(* IEC 61131-3 sources: ladder-web-ide/spikes/modelo/preset25, 22 files *)

(* ---- variante_a_pv13_base.st ---- *)
(* Variante A -- BASELINE do preset25 (spikes/modelo/NOTAS.md, "Experimento
   BLINK"). E o mesmo desenho/ST de spikes/modelo/blink_ladder.st (PV=13),
   reproduzido aqui como ponto de partida da matriz, para todas as variantes
   ficarem juntas e serem medidas pelo mesmo medir.py. Ver RESULTADO.md para
   a tabela comparativa.

   Ladder (ASCII; "%" = ramo paralelo na linha 1):

   Rung 1 (pulso, oscilador de 1 ciclo):
   ====|/pulso|==================( pulso )====

   Rung 2 (contador):
   ====|pulso|===+==[ CTU PV=13 ]===saida=atingiu====
                 %
                 +--|reset_ctu|--+   (ramo linha 1, alimenta R)

   Rung 3 (agenda reset, MINIMO de 1 ciclo de atraso -- e o proprio Q lido
           1 ciclo depois, por construcao: nao ha como um CTU usar seu
           proprio Q como R na MESMA chamada -- ver RESULTADO.md, prova):
   ====|atingiu|=================( reset_ctu )====

   Rung 4 (instantaneo de led, evita auto-cancelamento SET/RESET no mesmo
           scan -- ver NOTAS.md, "Risco descoberto no experimento"):
   ====|led|======================( led_estava_aceso )====

   Rung 5 (liga led):
   ====|atingiu|==|/led_estava_aceso|========(S led )====

   Rung 6 (desliga led):
   ====|atingiu|==|led_estava_aceso|=========(R led )====

   Rung 7 (botao, igual ao blink.st original):
   ====|botao|====================(S led )====

   ST derivado (ordem de leitura = ordem de execucao):
     pulso := NOT pulso;
     ctu0(CU := pulso, R := reset_ctu, PV := 13);
     atingiu := ctu0.Q;
     reset_ctu := atingiu;
     led_estava_aceso := led;
     IF atingiu AND NOT led_estava_aceso THEN led := TRUE; END_IF;
     IF atingiu AND led_estava_aceso THEN led := FALSE; END_IF;
     IF botao THEN led := TRUE; END_IF;

   Sem acentos: ASCII puro para o compilador. *)

PROGRAM prog0
  VAR
    botao AT %IX0.0 : BOOL;
    led   AT %QX0.0 : BOOL;
  END_VAR
  VAR
    pulso            : BOOL;
    reset_ctu        : BOOL;
    atingiu          : BOOL;
    led_estava_aceso : BOOL;
    ctu0             : CTU;
  END_VAR

  (* Rung 1 *)
  pulso := NOT pulso;

  (* Rung 2 *)
  ctu0(CU := pulso, R := reset_ctu, PV := 13);
  atingiu := ctu0.Q;

  (* Rung 3 -- reset com o atraso MINIMO possivel (1 scan) *)
  reset_ctu := atingiu;

  (* Rung 4 -- instantaneo de led *)
  led_estava_aceso := led;

  (* Rung 5 *)
  IF atingiu AND NOT led_estava_aceso THEN
    led := TRUE;
  END_IF;

  (* Rung 6 *)
  IF atingiu AND led_estava_aceso THEN
    led := FALSE;
  END_IF;

  (* Rung 7 *)
  IF botao THEN
    led := TRUE;
  END_IF;
END_PROGRAM

CONFIGURATION Config0
  RESOURCE Res0 ON PLC
    TASK task0(INTERVAL := T#20ms, PRIORITY := 0);
    PROGRAM instance0 WITH task0 : prog0;
  END_RESOURCE
END_CONFIGURATION

(* ---- variante_b_pv12.st ---- *)
(* Variante B -- mesmo desenho da variante A, PV=12 em vez de 13 (mesma
   tentativa "PV diferente" ja medida em spikes/modelo/blink_ladder_pv12.st,
   reproduzida aqui para entrar na mesma bateria de medicao de 200 ciclos /
   3 padroes de %IX0.0 do preset25). Ver RESULTADO.md.

   Ladder identico ao da variante A (variante_a_pv13_base.st), so troca
   PV:=13 por PV:=12 no rung 2. ST derivado idem, com PV:=12. *)

PROGRAM prog0
  VAR
    botao AT %IX0.0 : BOOL;
    led   AT %QX0.0 : BOOL;
  END_VAR
  VAR
    pulso            : BOOL;
    reset_ctu        : BOOL;
    atingiu          : BOOL;
    led_estava_aceso : BOOL;
    ctu0             : CTU;
  END_VAR

  (* Rung 1 *)
  pulso := NOT pulso;

  (* Rung 2 -- unica diferenca frente a variante A: PV=12 *)
  ctu0(CU := pulso, R := reset_ctu, PV := 12);
  atingiu := ctu0.Q;

  (* Rung 3 *)
  reset_ctu := atingiu;

  (* Rung 4 *)
  led_estava_aceso := led;

  (* Rung 5 *)
  IF atingiu AND NOT led_estava_aceso THEN
    led := TRUE;
  END_IF;

  (* Rung 6 *)
  IF atingiu AND led_estava_aceso THEN
    led := FALSE;
  END_IF;

  (* Rung 7 *)
  IF botao THEN
    led := TRUE;
  END_IF;
END_PROGRAM

CONFIGURATION Config0
  RESOURCE Res0 ON PLC
    TASK task0(INTERVAL := T#20ms, PRIORITY := 0);
    PROGRAM instance0 WITH task0 : prog0;
  END_RESOURCE
END_CONFIGURATION

(* ---- variante_c_pv25.st ---- *)
(* Variante C -- mesmo desenho da variante A, PV=25 (o valor "obvio" -- PV
   igual ao limite de contador.st -- citado no enunciado como tentativa a
   medir). Previsao analitica (RESULTADO.md, prova do periodo minimo
   T=2*PV): com CU alternando 1 vez por ciclo (borda a cada 2 ciclos) e reset
   consumindo 1 ciclo, o periodo minimo entre disparos de `atingiu` e
   2*25=50 ciclos -- 2x mais lento que os 25 ciclos de blink.st, nao um
   candidato melhor que PV=13. Medido aqui para confirmar. *)

PROGRAM prog0
  VAR
    botao AT %IX0.0 : BOOL;
    led   AT %QX0.0 : BOOL;
  END_VAR
  VAR
    pulso            : BOOL;
    reset_ctu        : BOOL;
    atingiu          : BOOL;
    led_estava_aceso : BOOL;
    ctu0             : CTU;
  END_VAR

  (* Rung 1 *)
  pulso := NOT pulso;

  (* Rung 2 -- unica diferenca frente a variante A: PV=25 *)
  ctu0(CU := pulso, R := reset_ctu, PV := 25);
  atingiu := ctu0.Q;

  (* Rung 3 *)
  reset_ctu := atingiu;

  (* Rung 4 *)
  led_estava_aceso := led;

  (* Rung 5 *)
  IF atingiu AND NOT led_estava_aceso THEN
    led := TRUE;
  END_IF;

  (* Rung 6 *)
  IF atingiu AND led_estava_aceso THEN
    led := FALSE;
  END_IF;

  (* Rung 7 *)
  IF botao THEN
    led := TRUE;
  END_IF;
END_PROGRAM

CONFIGURATION Config0
  RESOURCE Res0 ON PLC
    TASK task0(INTERVAL := T#20ms, PRIORITY := 0);
    PROGRAM instance0 WITH task0 : prog0;
  END_RESOURCE
END_CONFIGURATION

(* ---- variante_d_pv13_reset_atrasado.st ---- *)
(* Variante D -- PV=13, reset com 1 ciclo de atraso EXTRA (2 scans no total,
   em vez do minimo de 1 -- ver variante A) frente ao momento em que
   `atingiu` fica verdadeiro. Testa a celula da matriz "reset imediato
   (minimo possivel, variante A) vs atrasado" pedida no enunciado.

   Para conseguir um segundo scan de atraso sem tocar no elemento `ctu` (que
   so aceita R vindo de um caminho de contatos), uso DOIS estagios de
   bobina -- mas a ORDEM dos rungs importa (isto foi corrigido depois de
   medir: a primeira versao desta variante, com os dois rungs na ordem
   "contrario", nao acrescentava atraso nenhum -- ver NOTA DE MEDICAO no
   fim deste comentario):

     Rung 3 (ANTES do estagio 1): reset_ctu := reset_estagio1
       -- le reset_estagio1 como estava NO INICIO deste scan (o rung
       seguinte ainda nao o atualizou), ou seja o valor que o rung 4
       escreveu no scan ANTERIOR.
     Rung 4 (DEPOIS): reset_estagio1 := atingiu
       -- atualiza com o `atingiu` fresco deste mesmo scan.

   Com essa ordem: reset_estagio1(n) = atingiu(n); reset_ctu(n) =
   reset_estagio1(n-1) [valor pre-atualizacao] = atingiu(n-1). O `R` usado
   pela chamada do CTU no scan n+1 e reset_ctu(n) = atingiu(n-1) -- 2 scans
   de atraso frente a atingiu(n), 1 scan a mais que a variante A (que da
   R(n+1) = atingiu(n)).

   Ladder (ASCII):

   Rung 1 (pulso):
   ====|/pulso|==================( pulso )====

   Rung 2 (contador, mesmo desenho da variante A):
   ====|pulso|===+==[ CTU PV=13 ]===saida=atingiu====
                 %
                 +--|reset_ctu|--+

   Rung 3 (le o estagio 1 ANTES dele ser atualizado neste mesmo scan --
           e o que da o segundo scan de atraso):
   ====|reset_estagio1|===========( reset_ctu )====

   Rung 4 (so agora atualiza o estagio 1 com o `atingiu` fresco):
   ====|atingiu|=================( reset_estagio1 )====

   Rung 5 (instantaneo de led, igual a variante A):
   ====|led|======================( led_estava_aceso )====

   Rung 6 (liga led):
   ====|atingiu|==|/led_estava_aceso|========(S led )====

   Rung 7 (desliga led):
   ====|atingiu|==|led_estava_aceso|=========(R led )====

   Rung 8 (botao):
   ====|botao|====================(S led )====

   ST derivado:
     pulso := NOT pulso;
     ctu0(CU := pulso, R := reset_ctu, PV := 13);
     atingiu := ctu0.Q;
     reset_ctu := reset_estagio1;
     reset_estagio1 := atingiu;
     led_estava_aceso := led;
     IF atingiu AND NOT led_estava_aceso THEN led := TRUE; END_IF;
     IF atingiu AND led_estava_aceso THEN led := FALSE; END_IF;
     IF botao THEN led := TRUE; END_IF;

   NOTA DE MEDICAO (achado no proprio processo de montar esta variante, nao
   so no experimento original): a primeira tentativa de escrever este atraso
   extra colocou "reset_estagio1 := atingiu" ANTES de "reset_ctu :=
   reset_estagio1", isto e, deixou o valor fresco de `atingiu` atravessar os
   dois estagios NO MESMO SCAN (rung3 grava reset_estagio1(n)=atingiu(n);
   rung4, logo em seguida, ja le esse valor fresco e grava
   reset_ctu(n)=atingiu(n) -- zero atraso ADICIONAL, resultado identico ao
   da variante A). So a ordem escrita acima (ler o estagio seguinte ANTES de
   atualizar o anterior) de fato empurra 1 scan a mais -- e a mesma logica,
   inversa, de por que a variante A ja e o atraso MINIMO possivel (rung do
   reset depois do rung do CTU): o numero de scans de atraso de uma cadeia
   de bobinas depende de QUAL lado da cadeia e lido antes do outro ser
   escrito, nao so de quantos estagios existem. Medido com medir.py: a
   PRIMEIRA versao (sem atraso extra de fato) deu os MESMOS 22/22/21
   divergencias da variante A; esta versao corrigida e a que aparece na
   tabela de RESULTADO.md como "variante D". *)

PROGRAM prog0
  VAR
    botao AT %IX0.0 : BOOL;
    led   AT %QX0.0 : BOOL;
  END_VAR
  VAR
    pulso            : BOOL;
    reset_estagio1   : BOOL;
    reset_ctu        : BOOL;
    atingiu          : BOOL;
    led_estava_aceso : BOOL;
    ctu0             : CTU;
  END_VAR

  (* Rung 1 *)
  pulso := NOT pulso;

  (* Rung 2 *)
  ctu0(CU := pulso, R := reset_ctu, PV := 13);
  atingiu := ctu0.Q;

  (* Rung 3 -- le reset_estagio1 ANTES do rung 4 atualiza-lo (2o scan de atraso) *)
  reset_ctu := reset_estagio1;

  (* Rung 4 -- so agora atualiza com o atingiu fresco deste scan *)
  reset_estagio1 := atingiu;

  (* Rung 5 *)
  led_estava_aceso := led;

  (* Rung 6 *)
  IF atingiu AND NOT led_estava_aceso THEN
    led := TRUE;
  END_IF;

  (* Rung 7 *)
  IF atingiu AND led_estava_aceso THEN
    led := FALSE;
  END_IF;

  (* Rung 8 *)
  IF botao THEN
    led := TRUE;
  END_IF;
END_PROGRAM

CONFIGURATION Config0
  RESOURCE Res0 ON PLC
    TASK task0(INTERVAL := T#20ms, PRIORITY := 0);
    PROGRAM instance0 WITH task0 : prog0;
  END_RESOURCE
END_CONFIGURATION

(* ---- variante_e_pv13_toggle_paralelo.st ---- *)
(* Variante E -- PV=13, mesmo contador da variante A, mas o `led` alterna
   por um UNICO rung combinacional (ramo paralelo), nao por par SET/RESET.
   Testa a celula da matriz "toggle por ramo paralelo com bobina simples:
   led := (atingiu AND NOT led) OR (NOT atingiu AND led)".

   Motivo de interesse independente da fase: este desenho substitui os
   rungs 4/5/6 da variante A (instantaneo + par SET/RESET) por 1 rung so,
   eliminando de saida o risco de auto-cancelamento no mesmo scan descrito
   em NOTAS.md (nao ha dois rungs escrevendo o mesmo bit no mesmo scan) --
   `led_estava_aceso` deixa de ser necessario. Verifica-se aqui se isso muda
   a contagem/posicao das divergencias de fase (nao deveria: e uma troca de
   MECANISMO de toggle, nao do periodo do CTU).

   Ladder (ASCII):

   Rung 1 (pulso):
   ====|/pulso|==================( pulso )====

   Rung 2 (contador, igual a variante A):
   ====|pulso|===+==[ CTU PV=13 ]===saida=atingiu====
                 %
                 +--|reset_ctu|--+

   Rung 3 (agenda reset, igual a variante A):
   ====|atingiu|=================( reset_ctu )====

   Rung 4 (toggle combinacional -- DOIS caminhos em paralelo que se juntam
           na mesma bobina `led`; nenhum SET/RESET):
   ====|atingiu|==|/led|====+==================( led )====
   ====|/atingiu|==|led|====+

   Rung 5 (botao, igual a variante A):
   ====|botao|====================(S led )====

   ST derivado (a bobina comum de um rung com ramo paralelo e o OU dos
   caminhos serie -- aqui exatamente a expressao do enunciado):
     pulso := NOT pulso;
     ctu0(CU := pulso, R := reset_ctu, PV := 13);
     atingiu := ctu0.Q;
     reset_ctu := atingiu;
     led := (atingiu AND NOT led) OR (NOT atingiu AND led);
     IF botao THEN led := TRUE; END_IF; *)

PROGRAM prog0
  VAR
    botao AT %IX0.0 : BOOL;
    led   AT %QX0.0 : BOOL;
  END_VAR
  VAR
    pulso     : BOOL;
    reset_ctu : BOOL;
    atingiu   : BOOL;
    ctu0      : CTU;
  END_VAR

  (* Rung 1 *)
  pulso := NOT pulso;

  (* Rung 2 *)
  ctu0(CU := pulso, R := reset_ctu, PV := 13);
  atingiu := ctu0.Q;

  (* Rung 3 *)
  reset_ctu := atingiu;

  (* Rung 4 -- toggle por ramo paralelo, sem SET/RESET *)
  led := (atingiu AND NOT led) OR (NOT atingiu AND led);

  (* Rung 5 *)
  IF botao THEN
    led := TRUE;
  END_IF;
END_PROGRAM

CONFIGURATION Config0
  RESOURCE Res0 ON PLC
    TASK task0(INTERVAL := T#20ms, PRIORITY := 0);
    PROGRAM instance0 WITH task0 : prog0;
  END_RESOURCE
END_CONFIGURATION

(* ---- variante_f_pv13_pulso_inicial_true.st ---- *)
(* Variante F -- PV=13, mesmo desenho da variante A, so muda o valor
   INICIAL de `pulso` para TRUE em vez do default FALSE. Testa a celula da
   matriz "pulso inicial FALSE/TRUE".

   ACHADO A REGISTRAR (ver RESULTADO.md): o modelo grafico obrigatorio
   (spikes/modelo/modelo.ts, interface `Variavel`) NAO tem campo de valor
   inicial -- so `nome`, `tipo`, `endereco?`. Esta variante e expressavel em
   ST puro (`pulso : BOOL := TRUE;`, sintaxe valida de IEC 61131-3), mas NAO
   e desenhavel com o modelo de dados da grade tal como ele existe hoje: um
   editor Ladder que use esse modelo nao tem como o autor do diagrama pedir
   "essa variavel comeca em TRUE". Se esta variante fosse a vencedora,
   `Variavel` precisaria ganhar um campo tipo `valorInicial?: boolean` (so
   faz sentido para BOOL nao localizado; UINT e localizado ficam fora). Ela
   NAO e a vencedora (ver RESULTADO.md), entao o gap fica soh registrado,
   sem exigir mudanca no modelo.

   Ladder: identico a variante A (nao ha elemento grafico que represente
   "valor inicial"; a diferenca so aparece no ST). *)

PROGRAM prog0
  VAR
    botao AT %IX0.0 : BOOL;
    led   AT %QX0.0 : BOOL;
  END_VAR
  VAR
    pulso            : BOOL := TRUE; (* unica diferenca frente a variante A *)
    reset_ctu        : BOOL;
    atingiu          : BOOL;
    led_estava_aceso : BOOL;
    ctu0             : CTU;
  END_VAR

  (* Rung 1 *)
  pulso := NOT pulso;

  (* Rung 2 *)
  ctu0(CU := pulso, R := reset_ctu, PV := 13);
  atingiu := ctu0.Q;

  (* Rung 3 *)
  reset_ctu := atingiu;

  (* Rung 4 *)
  led_estava_aceso := led;

  (* Rung 5 *)
  IF atingiu AND NOT led_estava_aceso THEN
    led := TRUE;
  END_IF;

  (* Rung 6 *)
  IF atingiu AND led_estava_aceso THEN
    led := FALSE;
  END_IF;

  (* Rung 7 *)
  IF botao THEN
    led := TRUE;
  END_IF;
END_PROGRAM

CONFIGURATION Config0
  RESOURCE Res0 ON PLC
    TASK task0(INTERVAL := T#20ms, PRIORITY := 0);
    PROGRAM instance0 WITH task0 : prog0;
  END_RESOURCE
END_CONFIGURATION

(* ---- variante_g_pv13_ordem_invertida.st ---- *)
(* Variante G -- PV=13, mesmo desenho da variante A, mas o rung do CTU vem
   ANTES do rung que alterna `pulso` (ordem de leitura trocada). Testa a
   celula da matriz "rung de pulso antes/depois do rung do CTU".

   Com essa troca, o `CU` que o CTU le no scan N e o `pulso` como ficou no
   FIM do scan N-1 (o toggle deste scan so acontece DEPOIS, no rung
   seguinte) -- desloca a fase de leitura de `pulso` em 1 scan frente a
   variante A, analogo ao que um valor inicial diferente faria, mas via
   ordem de rung em vez de valor inicial (essa SIM e desenhavel no modelo
   grafico hoje: e so por o rung do contador antes do rung do oscilador na
   lista `rungs` do `Diagrama` -- nao exige nenhum campo novo).

   Ladder (ASCII; ordem trocada frente a variante A):

   Rung 1 (contador, agora primeiro):
   ====|pulso|===+==[ CTU PV=13 ]===saida=atingiu====
                 %
                 +--|reset_ctu|--+

   Rung 2 (pulso, agora depois):
   ====|/pulso|==================( pulso )====

   Rung 3 (agenda reset):
   ====|atingiu|=================( reset_ctu )====

   Rung 4 (instantaneo de led):
   ====|led|======================( led_estava_aceso )====

   Rung 5 (liga led):
   ====|atingiu|==|/led_estava_aceso|========(S led )====

   Rung 6 (desliga led):
   ====|atingiu|==|led_estava_aceso|=========(R led )====

   Rung 7 (botao):
   ====|botao|====================(S led )====

   ST derivado (so a ordem das duas primeiras atribuicoes muda frente a
   variante A):
     ctu0(CU := pulso, R := reset_ctu, PV := 13);
     atingiu := ctu0.Q;
     pulso := NOT pulso;
     reset_ctu := atingiu;
     led_estava_aceso := led;
     IF atingiu AND NOT led_estava_aceso THEN led := TRUE; END_IF;
     IF atingiu AND led_estava_aceso THEN led := FALSE; END_IF;
     IF botao THEN led := TRUE; END_IF; *)

PROGRAM prog0
  VAR
    botao AT %IX0.0 : BOOL;
    led   AT %QX0.0 : BOOL;
  END_VAR
  VAR
    pulso            : BOOL;
    reset_ctu        : BOOL;
    atingiu          : BOOL;
    led_estava_aceso : BOOL;
    ctu0             : CTU;
  END_VAR

  (* Rung 1 -- contador, ANTES do toggle de pulso (ordem trocada) *)
  ctu0(CU := pulso, R := reset_ctu, PV := 13);
  atingiu := ctu0.Q;

  (* Rung 2 -- pulso, agora depois *)
  pulso := NOT pulso;

  (* Rung 3 *)
  reset_ctu := atingiu;

  (* Rung 4 *)
  led_estava_aceso := led;

  (* Rung 5 *)
  IF atingiu AND NOT led_estava_aceso THEN
    led := TRUE;
  END_IF;

  (* Rung 6 *)
  IF atingiu AND led_estava_aceso THEN
    led := FALSE;
  END_IF;

  (* Rung 7 *)
  IF botao THEN
    led := TRUE;
  END_IF;
END_PROGRAM

CONFIGURATION Config0
  RESOURCE Res0 ON PLC
    TASK task0(INTERVAL := T#20ms, PRIORITY := 0);
    PROGRAM instance0 WITH task0 : prog0;
  END_RESOURCE
END_CONFIGURATION

(* ---- variante_h_pv12_reset_atrasado.st ---- *)
(* Variante D -- PV=13, reset com 1 ciclo de atraso EXTRA (2 scans no total,
   em vez do minimo de 1 -- ver variante A) frente ao momento em que
   `atingiu` fica verdadeiro. Testa a celula da matriz "reset imediato
   (minimo possivel, variante A) vs atrasado" pedida no enunciado.

   Para conseguir um segundo scan de atraso sem tocar no elemento `ctu` (que
   so aceita R vindo de um caminho de contatos), uso DOIS estagios de
   bobina -- mas a ORDEM dos rungs importa (isto foi corrigido depois de
   medir: a primeira versao desta variante, com os dois rungs na ordem
   "contrario", nao acrescentava atraso nenhum -- ver NOTA DE MEDICAO no
   fim deste comentario):

     Rung 3 (ANTES do estagio 1): reset_ctu := reset_estagio1
       -- le reset_estagio1 como estava NO INICIO deste scan (o rung
       seguinte ainda nao o atualizou), ou seja o valor que o rung 4
       escreveu no scan ANTERIOR.
     Rung 4 (DEPOIS): reset_estagio1 := atingiu
       -- atualiza com o `atingiu` fresco deste mesmo scan.

   Com essa ordem: reset_estagio1(n) = atingiu(n); reset_ctu(n) =
   reset_estagio1(n-1) [valor pre-atualizacao] = atingiu(n-1). O `R` usado
   pela chamada do CTU no scan n+1 e reset_ctu(n) = atingiu(n-1) -- 2 scans
   de atraso frente a atingiu(n), 1 scan a mais que a variante A (que da
   R(n+1) = atingiu(n)).

   Ladder (ASCII):

   Rung 1 (pulso):
   ====|/pulso|==================( pulso )====

   Rung 2 (contador, mesmo desenho da variante A):
   ====|pulso|===+==[ CTU PV=13 ]===saida=atingiu====
                 %
                 +--|reset_ctu|--+

   Rung 3 (le o estagio 1 ANTES dele ser atualizado neste mesmo scan --
           e o que da o segundo scan de atraso):
   ====|reset_estagio1|===========( reset_ctu )====

   Rung 4 (so agora atualiza o estagio 1 com o `atingiu` fresco):
   ====|atingiu|=================( reset_estagio1 )====

   Rung 5 (instantaneo de led, igual a variante A):
   ====|led|======================( led_estava_aceso )====

   Rung 6 (liga led):
   ====|atingiu|==|/led_estava_aceso|========(S led )====

   Rung 7 (desliga led):
   ====|atingiu|==|led_estava_aceso|=========(R led )====

   Rung 8 (botao):
   ====|botao|====================(S led )====

   ST derivado:
     pulso := NOT pulso;
     ctu0(CU := pulso, R := reset_ctu, PV := 12);
     atingiu := ctu0.Q;
     reset_ctu := reset_estagio1;
     reset_estagio1 := atingiu;
     led_estava_aceso := led;
     IF atingiu AND NOT led_estava_aceso THEN led := TRUE; END_IF;
     IF atingiu AND led_estava_aceso THEN led := FALSE; END_IF;
     IF botao THEN led := TRUE; END_IF;

   NOTA DE MEDICAO (achado no proprio processo de montar esta variante, nao
   so no experimento original): a primeira tentativa de escrever este atraso
   extra colocou "reset_estagio1 := atingiu" ANTES de "reset_ctu :=
   reset_estagio1", isto e, deixou o valor fresco de `atingiu` atravessar os
   dois estagios NO MESMO SCAN (rung3 grava reset_estagio1(n)=atingiu(n);
   rung4, logo em seguida, ja le esse valor fresco e grava
   reset_ctu(n)=atingiu(n) -- zero atraso ADICIONAL, resultado identico ao
   da variante A). So a ordem escrita acima (ler o estagio seguinte ANTES de
   atualizar o anterior) de fato empurra 1 scan a mais -- e a mesma logica,
   inversa, de por que a variante A ja e o atraso MINIMO possivel (rung do
   reset depois do rung do CTU): o numero de scans de atraso de uma cadeia
   de bobinas depende de QUAL lado da cadeia e lido antes do outro ser
   escrito, nao so de quantos estagios existem. Medido com medir.py: a
   PRIMEIRA versao (sem atraso extra de fato) deu os MESMOS 22/22/21
   divergencias da variante A; esta versao corrigida e a que aparece na
   tabela de RESULTADO.md como "variante D". *)

PROGRAM prog0
  VAR
    botao AT %IX0.0 : BOOL;
    led   AT %QX0.0 : BOOL;
  END_VAR
  VAR
    pulso            : BOOL;
    reset_estagio1   : BOOL;
    reset_ctu        : BOOL;
    atingiu          : BOOL;
    led_estava_aceso : BOOL;
    ctu0             : CTU;
  END_VAR

  (* Rung 1 *)
  pulso := NOT pulso;

  (* Rung 2 *)
  ctu0(CU := pulso, R := reset_ctu, PV := 12);
  atingiu := ctu0.Q;

  (* Rung 3 -- le reset_estagio1 ANTES do rung 4 atualiza-lo (2o scan de atraso) *)
  reset_ctu := reset_estagio1;

  (* Rung 4 -- so agora atualiza com o atingiu fresco deste scan *)
  reset_estagio1 := atingiu;

  (* Rung 5 *)
  led_estava_aceso := led;

  (* Rung 6 *)
  IF atingiu AND NOT led_estava_aceso THEN
    led := TRUE;
  END_IF;

  (* Rung 7 *)
  IF atingiu AND led_estava_aceso THEN
    led := FALSE;
  END_IF;

  (* Rung 8 *)
  IF botao THEN
    led := TRUE;
  END_IF;
END_PROGRAM

CONFIGURATION Config0
  RESOURCE Res0 ON PLC
    TASK task0(INTERVAL := T#20ms, PRIORITY := 0);
    PROGRAM instance0 WITH task0 : prog0;
  END_RESOURCE
END_CONFIGURATION

(* ---- variante_i_pv12_reset_pulso.st ---- *)
(* Variante A -- BASELINE do preset25 (spikes/modelo/NOTAS.md, "Experimento
   BLINK"). E o mesmo desenho/ST de spikes/modelo/blink_ladder.st (PV=13),
   reproduzido aqui como ponto de partida da matriz, para todas as variantes
   ficarem juntas e serem medidas pelo mesmo medir.py. Ver RESULTADO.md para
   a tabela comparativa.

   Ladder (ASCII; "%" = ramo paralelo na linha 1):

   Rung 1 (pulso, oscilador de 1 ciclo):
   ====|/pulso|==================( pulso )====

   Rung 2 (contador):
   ====|pulso|===+==[ CTU PV=13 ]===saida=atingiu====
                 %
                 +--|reset_ctu|--+   (ramo linha 1, alimenta R)

   Rung 3 (agenda reset, MINIMO de 1 ciclo de atraso -- e o proprio Q lido
           1 ciclo depois, por construcao: nao ha como um CTU usar seu
           proprio Q como R na MESMA chamada -- ver RESULTADO.md, prova):
   ====|atingiu|=================( reset_ctu )====

   Rung 4 (instantaneo de led, evita auto-cancelamento SET/RESET no mesmo
           scan -- ver NOTAS.md, "Risco descoberto no experimento"):
   ====|led|======================( led_estava_aceso )====

   Rung 5 (liga led):
   ====|atingiu|==|/led_estava_aceso|========(S led )====

   Rung 6 (desliga led):
   ====|atingiu|==|led_estava_aceso|=========(R led )====

   Rung 7 (botao, igual ao blink.st original):
   ====|botao|====================(S led )====

   ST derivado (ordem de leitura = ordem de execucao):
     pulso := NOT pulso;
     ctu0(CU := pulso, R := reset_ctu, PV := 12);
     atingiu := ctu0.Q;
     reset_ctu := atingiu;
     led_estava_aceso := led;
     IF atingiu AND NOT led_estava_aceso THEN led := TRUE; END_IF;
     IF atingiu AND led_estava_aceso THEN led := FALSE; END_IF;
     IF botao THEN led := TRUE; END_IF;

   Sem acentos: ASCII puro para o compilador. *)

PROGRAM prog0
  VAR
    botao AT %IX0.0 : BOOL;
    led   AT %QX0.0 : BOOL;
  END_VAR
  VAR
    pulso            : BOOL;
    reset_ctu        : BOOL;
    atingiu          : BOOL;
    led_estava_aceso : BOOL;
    ctu0             : CTU;
  END_VAR

  (* Rung 1 *)
  pulso := NOT pulso;

  (* Rung 2 *)
  ctu0(CU := pulso, R := reset_ctu, PV := 12);
  atingiu := ctu0.Q;

  (* Rung 2b -- reset de pulso ao atingir: realinha a grade de bordas *)
  IF atingiu THEN
    pulso := FALSE;
  END_IF;

  (* Rung 3 -- reset com o atraso MINIMO possivel (1 scan) *)
  reset_ctu := atingiu;

  (* Rung 4 -- instantaneo de led *)
  led_estava_aceso := led;

  (* Rung 5 *)
  IF atingiu AND NOT led_estava_aceso THEN
    led := TRUE;
  END_IF;

  (* Rung 6 *)
  IF atingiu AND led_estava_aceso THEN
    led := FALSE;
  END_IF;

  (* Rung 7 *)
  IF botao THEN
    led := TRUE;
  END_IF;
END_PROGRAM

CONFIGURATION Config0
  RESOURCE Res0 ON PLC
    TASK task0(INTERVAL := T#20ms, PRIORITY := 0);
    PROGRAM instance0 WITH task0 : prog0;
  END_RESOURCE
END_CONFIGURATION

(* ---- variante_i_pv12_set_pulso.st ---- *)
(* Variante A -- BASELINE do preset25 (spikes/modelo/NOTAS.md, "Experimento
   BLINK"). E o mesmo desenho/ST de spikes/modelo/blink_ladder.st (PV=13),
   reproduzido aqui como ponto de partida da matriz, para todas as variantes
   ficarem juntas e serem medidas pelo mesmo medir.py. Ver RESULTADO.md para
   a tabela comparativa.

   Ladder (ASCII; "%" = ramo paralelo na linha 1):

   Rung 1 (pulso, oscilador de 1 ciclo):
   ====|/pulso|==================( pulso )====

   Rung 2 (contador):
   ====|pulso|===+==[ CTU PV=13 ]===saida=atingiu====
                 %
                 +--|reset_ctu|--+   (ramo linha 1, alimenta R)

   Rung 3 (agenda reset, MINIMO de 1 ciclo de atraso -- e o proprio Q lido
           1 ciclo depois, por construcao: nao ha como um CTU usar seu
           proprio Q como R na MESMA chamada -- ver RESULTADO.md, prova):
   ====|atingiu|=================( reset_ctu )====

   Rung 4 (instantaneo de led, evita auto-cancelamento SET/RESET no mesmo
           scan -- ver NOTAS.md, "Risco descoberto no experimento"):
   ====|led|======================( led_estava_aceso )====

   Rung 5 (liga led):
   ====|atingiu|==|/led_estava_aceso|========(S led )====

   Rung 6 (desliga led):
   ====|atingiu|==|led_estava_aceso|=========(R led )====

   Rung 7 (botao, igual ao blink.st original):
   ====|botao|====================(S led )====

   ST derivado (ordem de leitura = ordem de execucao):
     pulso := NOT pulso;
     ctu0(CU := pulso, R := reset_ctu, PV := 12);
     atingiu := ctu0.Q;
     reset_ctu := atingiu;
     led_estava_aceso := led;
     IF atingiu AND NOT led_estava_aceso THEN led := TRUE; END_IF;
     IF atingiu AND led_estava_aceso THEN led := FALSE; END_IF;
     IF botao THEN led := TRUE; END_IF;

   Sem acentos: ASCII puro para o compilador. *)

PROGRAM prog0
  VAR
    botao AT %IX0.0 : BOOL;
    led   AT %QX0.0 : BOOL;
  END_VAR
  VAR
    pulso            : BOOL;
    reset_ctu        : BOOL;
    atingiu          : BOOL;
    led_estava_aceso : BOOL;
    ctu0             : CTU;
  END_VAR

  (* Rung 1 *)
  pulso := NOT pulso;

  (* Rung 2 *)
  ctu0(CU := pulso, R := reset_ctu, PV := 12);
  atingiu := ctu0.Q;

  (* Rung 2b -- set de pulso ao atingir: realinha a grade de bordas *)
  IF atingiu THEN
    pulso := TRUE;
  END_IF;

  (* Rung 3 -- reset com o atraso MINIMO possivel (1 scan) *)
  reset_ctu := atingiu;

  (* Rung 4 -- instantaneo de led *)
  led_estava_aceso := led;

  (* Rung 5 *)
  IF atingiu AND NOT led_estava_aceso THEN
    led := TRUE;
  END_IF;

  (* Rung 6 *)
  IF atingiu AND led_estava_aceso THEN
    led := FALSE;
  END_IF;

  (* Rung 7 *)
  IF botao THEN
    led := TRUE;
  END_IF;
END_PROGRAM

CONFIGURATION Config0
  RESOURCE Res0 ON PLC
    TASK task0(INTERVAL := T#20ms, PRIORITY := 0);
    PROGRAM instance0 WITH task0 : prog0;
  END_RESOURCE
END_CONFIGURATION

(* ---- variante_i_pv13_reset_pulso.st ---- *)
(* Variante A -- BASELINE do preset25 (spikes/modelo/NOTAS.md, "Experimento
   BLINK"). E o mesmo desenho/ST de spikes/modelo/blink_ladder.st (PV=13),
   reproduzido aqui como ponto de partida da matriz, para todas as variantes
   ficarem juntas e serem medidas pelo mesmo medir.py. Ver RESULTADO.md para
   a tabela comparativa.

   Ladder (ASCII; "%" = ramo paralelo na linha 1):

   Rung 1 (pulso, oscilador de 1 ciclo):
   ====|/pulso|==================( pulso )====

   Rung 2 (contador):
   ====|pulso|===+==[ CTU PV=13 ]===saida=atingiu====
                 %
                 +--|reset_ctu|--+   (ramo linha 1, alimenta R)

   Rung 3 (agenda reset, MINIMO de 1 ciclo de atraso -- e o proprio Q lido
           1 ciclo depois, por construcao: nao ha como um CTU usar seu
           proprio Q como R na MESMA chamada -- ver RESULTADO.md, prova):
   ====|atingiu|=================( reset_ctu )====

   Rung 4 (instantaneo de led, evita auto-cancelamento SET/RESET no mesmo
           scan -- ver NOTAS.md, "Risco descoberto no experimento"):
   ====|led|======================( led_estava_aceso )====

   Rung 5 (liga led):
   ====|atingiu|==|/led_estava_aceso|========(S led )====

   Rung 6 (desliga led):
   ====|atingiu|==|led_estava_aceso|=========(R led )====

   Rung 7 (botao, igual ao blink.st original):
   ====|botao|====================(S led )====

   ST derivado (ordem de leitura = ordem de execucao):
     pulso := NOT pulso;
     ctu0(CU := pulso, R := reset_ctu, PV := 13);
     atingiu := ctu0.Q;
     reset_ctu := atingiu;
     led_estava_aceso := led;
     IF atingiu AND NOT led_estava_aceso THEN led := TRUE; END_IF;
     IF atingiu AND led_estava_aceso THEN led := FALSE; END_IF;
     IF botao THEN led := TRUE; END_IF;

   Sem acentos: ASCII puro para o compilador. *)

PROGRAM prog0
  VAR
    botao AT %IX0.0 : BOOL;
    led   AT %QX0.0 : BOOL;
  END_VAR
  VAR
    pulso            : BOOL;
    reset_ctu        : BOOL;
    atingiu          : BOOL;
    led_estava_aceso : BOOL;
    ctu0             : CTU;
  END_VAR

  (* Rung 1 *)
  pulso := NOT pulso;

  (* Rung 2 *)
  ctu0(CU := pulso, R := reset_ctu, PV := 13);
  atingiu := ctu0.Q;

  (* Rung 2b -- reset de pulso ao atingir: realinha a grade de bordas *)
  IF atingiu THEN
    pulso := FALSE;
  END_IF;

  (* Rung 3 -- reset com o atraso MINIMO possivel (1 scan) *)
  reset_ctu := atingiu;

  (* Rung 4 -- instantaneo de led *)
  led_estava_aceso := led;

  (* Rung 5 *)
  IF atingiu AND NOT led_estava_aceso THEN
    led := TRUE;
  END_IF;

  (* Rung 6 *)
  IF atingiu AND led_estava_aceso THEN
    led := FALSE;
  END_IF;

  (* Rung 7 *)
  IF botao THEN
    led := TRUE;
  END_IF;
END_PROGRAM

CONFIGURATION Config0
  RESOURCE Res0 ON PLC
    TASK task0(INTERVAL := T#20ms, PRIORITY := 0);
    PROGRAM instance0 WITH task0 : prog0;
  END_RESOURCE
END_CONFIGURATION

(* ---- variante_i_pv13_set_pulso.st ---- *)
(* Variante A -- BASELINE do preset25 (spikes/modelo/NOTAS.md, "Experimento
   BLINK"). E o mesmo desenho/ST de spikes/modelo/blink_ladder.st (PV=13),
   reproduzido aqui como ponto de partida da matriz, para todas as variantes
   ficarem juntas e serem medidas pelo mesmo medir.py. Ver RESULTADO.md para
   a tabela comparativa.

   Ladder (ASCII; "%" = ramo paralelo na linha 1):

   Rung 1 (pulso, oscilador de 1 ciclo):
   ====|/pulso|==================( pulso )====

   Rung 2 (contador):
   ====|pulso|===+==[ CTU PV=13 ]===saida=atingiu====
                 %
                 +--|reset_ctu|--+   (ramo linha 1, alimenta R)

   Rung 3 (agenda reset, MINIMO de 1 ciclo de atraso -- e o proprio Q lido
           1 ciclo depois, por construcao: nao ha como um CTU usar seu
           proprio Q como R na MESMA chamada -- ver RESULTADO.md, prova):
   ====|atingiu|=================( reset_ctu )====

   Rung 4 (instantaneo de led, evita auto-cancelamento SET/RESET no mesmo
           scan -- ver NOTAS.md, "Risco descoberto no experimento"):
   ====|led|======================( led_estava_aceso )====

   Rung 5 (liga led):
   ====|atingiu|==|/led_estava_aceso|========(S led )====

   Rung 6 (desliga led):
   ====|atingiu|==|led_estava_aceso|=========(R led )====

   Rung 7 (botao, igual ao blink.st original):
   ====|botao|====================(S led )====

   ST derivado (ordem de leitura = ordem de execucao):
     pulso := NOT pulso;
     ctu0(CU := pulso, R := reset_ctu, PV := 13);
     atingiu := ctu0.Q;
     reset_ctu := atingiu;
     led_estava_aceso := led;
     IF atingiu AND NOT led_estava_aceso THEN led := TRUE; END_IF;
     IF atingiu AND led_estava_aceso THEN led := FALSE; END_IF;
     IF botao THEN led := TRUE; END_IF;

   Sem acentos: ASCII puro para o compilador. *)

PROGRAM prog0
  VAR
    botao AT %IX0.0 : BOOL;
    led   AT %QX0.0 : BOOL;
  END_VAR
  VAR
    pulso            : BOOL;
    reset_ctu        : BOOL;
    atingiu          : BOOL;
    led_estava_aceso : BOOL;
    ctu0             : CTU;
  END_VAR

  (* Rung 1 *)
  pulso := NOT pulso;

  (* Rung 2 *)
  ctu0(CU := pulso, R := reset_ctu, PV := 13);
  atingiu := ctu0.Q;

  (* Rung 2b -- set de pulso ao atingir: realinha a grade de bordas *)
  IF atingiu THEN
    pulso := TRUE;
  END_IF;

  (* Rung 3 -- reset com o atraso MINIMO possivel (1 scan) *)
  reset_ctu := atingiu;

  (* Rung 4 -- instantaneo de led *)
  led_estava_aceso := led;

  (* Rung 5 *)
  IF atingiu AND NOT led_estava_aceso THEN
    led := TRUE;
  END_IF;

  (* Rung 6 *)
  IF atingiu AND led_estava_aceso THEN
    led := FALSE;
  END_IF;

  (* Rung 7 *)
  IF botao THEN
    led := TRUE;
  END_IF;
END_PROGRAM

CONFIGURATION Config0
  RESOURCE Res0 ON PLC
    TASK task0(INTERVAL := T#20ms, PRIORITY := 0);
    PROGRAM instance0 WITH task0 : prog0;
  END_RESOURCE
END_CONFIGURATION

(* ---- variante_j_pv12_ctu_antes_iniFALSE_realinhaFALSE.st ---- *)
(* Variante J (orquestrador, 2026-09-16): PV=12, pulso realinhado ao atingir o
   limite; ordem=ctu_antes, pulso inicial=FALSE, valor de realinhamento=FALSE. *)
PROGRAM prog0
  VAR
    botao AT %IX0.0 : BOOL;
    led   AT %QX0.0 : BOOL;
  END_VAR
  VAR
    pulso            : BOOL := FALSE;
    reset_ctu        : BOOL;
    atingiu          : BOOL;
    led_estava_aceso : BOOL;
    ctu0             : CTU;
  END_VAR

  ctu0(CU := pulso, R := reset_ctu, PV := 12);
  atingiu := ctu0.Q;
  IF atingiu THEN
    pulso := FALSE;
  END_IF;
  pulso := NOT pulso;
  reset_ctu := atingiu;
  led_estava_aceso := led;
  IF atingiu AND NOT led_estava_aceso THEN
    led := TRUE;
  END_IF;
  IF atingiu AND led_estava_aceso THEN
    led := FALSE;
  END_IF;
  IF botao THEN
    led := TRUE;
  END_IF;
END_PROGRAM

CONFIGURATION Config0
  RESOURCE Res0 ON PLC
    TASK task0(INTERVAL := T#20ms, PRIORITY := 0);
    PROGRAM instance0 WITH task0 : prog0;
  END_RESOURCE
END_CONFIGURATION

(* ---- variante_j_pv12_ctu_antes_iniFALSE_realinhaTRUE.st ---- *)
(* Variante J (orquestrador, 2026-09-16): PV=12, pulso realinhado ao atingir o
   limite; ordem=ctu_antes, pulso inicial=FALSE, valor de realinhamento=TRUE. *)
PROGRAM prog0
  VAR
    botao AT %IX0.0 : BOOL;
    led   AT %QX0.0 : BOOL;
  END_VAR
  VAR
    pulso            : BOOL := FALSE;
    reset_ctu        : BOOL;
    atingiu          : BOOL;
    led_estava_aceso : BOOL;
    ctu0             : CTU;
  END_VAR

  ctu0(CU := pulso, R := reset_ctu, PV := 12);
  atingiu := ctu0.Q;
  IF atingiu THEN
    pulso := TRUE;
  END_IF;
  pulso := NOT pulso;
  reset_ctu := atingiu;
  led_estava_aceso := led;
  IF atingiu AND NOT led_estava_aceso THEN
    led := TRUE;
  END_IF;
  IF atingiu AND led_estava_aceso THEN
    led := FALSE;
  END_IF;
  IF botao THEN
    led := TRUE;
  END_IF;
END_PROGRAM

CONFIGURATION Config0
  RESOURCE Res0 ON PLC
    TASK task0(INTERVAL := T#20ms, PRIORITY := 0);
    PROGRAM instance0 WITH task0 : prog0;
  END_RESOURCE
END_CONFIGURATION

(* ---- variante_j_pv12_ctu_antes_iniTRUE_realinhaFALSE.st ---- *)
(* Variante J (orquestrador, 2026-09-16): PV=12, pulso realinhado ao atingir o
   limite; ordem=ctu_antes, pulso inicial=TRUE, valor de realinhamento=FALSE. *)
PROGRAM prog0
  VAR
    botao AT %IX0.0 : BOOL;
    led   AT %QX0.0 : BOOL;
  END_VAR
  VAR
    pulso            : BOOL := TRUE;
    reset_ctu        : BOOL;
    atingiu          : BOOL;
    led_estava_aceso : BOOL;
    ctu0             : CTU;
  END_VAR

  ctu0(CU := pulso, R := reset_ctu, PV := 12);
  atingiu := ctu0.Q;
  IF atingiu THEN
    pulso := FALSE;
  END_IF;
  pulso := NOT pulso;
  reset_ctu := atingiu;
  led_estava_aceso := led;
  IF atingiu AND NOT led_estava_aceso THEN
    led := TRUE;
  END_IF;
  IF atingiu AND led_estava_aceso THEN
    led := FALSE;
  END_IF;
  IF botao THEN
    led := TRUE;
  END_IF;
END_PROGRAM

CONFIGURATION Config0
  RESOURCE Res0 ON PLC
    TASK task0(INTERVAL := T#20ms, PRIORITY := 0);
    PROGRAM instance0 WITH task0 : prog0;
  END_RESOURCE
END_CONFIGURATION

(* ---- variante_j_pv12_ctu_antes_iniTRUE_realinhaTRUE.st ---- *)
(* Variante J (orquestrador, 2026-09-16): PV=12, pulso realinhado ao atingir o
   limite; ordem=ctu_antes, pulso inicial=TRUE, valor de realinhamento=TRUE. *)
PROGRAM prog0
  VAR
    botao AT %IX0.0 : BOOL;
    led   AT %QX0.0 : BOOL;
  END_VAR
  VAR
    pulso            : BOOL := TRUE;
    reset_ctu        : BOOL;
    atingiu          : BOOL;
    led_estava_aceso : BOOL;
    ctu0             : CTU;
  END_VAR

  ctu0(CU := pulso, R := reset_ctu, PV := 12);
  atingiu := ctu0.Q;
  IF atingiu THEN
    pulso := TRUE;
  END_IF;
  pulso := NOT pulso;
  reset_ctu := atingiu;
  led_estava_aceso := led;
  IF atingiu AND NOT led_estava_aceso THEN
    led := TRUE;
  END_IF;
  IF atingiu AND led_estava_aceso THEN
    led := FALSE;
  END_IF;
  IF botao THEN
    led := TRUE;
  END_IF;
END_PROGRAM

CONFIGURATION Config0
  RESOURCE Res0 ON PLC
    TASK task0(INTERVAL := T#20ms, PRIORITY := 0);
    PROGRAM instance0 WITH task0 : prog0;
  END_RESOURCE
END_CONFIGURATION

(* ---- variante_j_pv12_pulso_antes_iniFALSE_realinhaFALSE.st ---- *)
(* Variante J (orquestrador, 2026-09-16): PV=12, pulso realinhado ao atingir o
   limite; ordem=pulso_antes, pulso inicial=FALSE, valor de realinhamento=FALSE. *)
PROGRAM prog0
  VAR
    botao AT %IX0.0 : BOOL;
    led   AT %QX0.0 : BOOL;
  END_VAR
  VAR
    pulso            : BOOL := FALSE;
    reset_ctu        : BOOL;
    atingiu          : BOOL;
    led_estava_aceso : BOOL;
    ctu0             : CTU;
  END_VAR

  pulso := NOT pulso;
  ctu0(CU := pulso, R := reset_ctu, PV := 12);
  atingiu := ctu0.Q;
  IF atingiu THEN
    pulso := FALSE;
  END_IF;
  reset_ctu := atingiu;
  led_estava_aceso := led;
  IF atingiu AND NOT led_estava_aceso THEN
    led := TRUE;
  END_IF;
  IF atingiu AND led_estava_aceso THEN
    led := FALSE;
  END_IF;
  IF botao THEN
    led := TRUE;
  END_IF;
END_PROGRAM

CONFIGURATION Config0
  RESOURCE Res0 ON PLC
    TASK task0(INTERVAL := T#20ms, PRIORITY := 0);
    PROGRAM instance0 WITH task0 : prog0;
  END_RESOURCE
END_CONFIGURATION

(* ---- variante_j_pv12_pulso_antes_iniFALSE_realinhaTRUE.st ---- *)
(* Variante J (orquestrador, 2026-09-16): PV=12, pulso realinhado ao atingir o
   limite; ordem=pulso_antes, pulso inicial=FALSE, valor de realinhamento=TRUE. *)
PROGRAM prog0
  VAR
    botao AT %IX0.0 : BOOL;
    led   AT %QX0.0 : BOOL;
  END_VAR
  VAR
    pulso            : BOOL := FALSE;
    reset_ctu        : BOOL;
    atingiu          : BOOL;
    led_estava_aceso : BOOL;
    ctu0             : CTU;
  END_VAR

  pulso := NOT pulso;
  ctu0(CU := pulso, R := reset_ctu, PV := 12);
  atingiu := ctu0.Q;
  IF atingiu THEN
    pulso := TRUE;
  END_IF;
  reset_ctu := atingiu;
  led_estava_aceso := led;
  IF atingiu AND NOT led_estava_aceso THEN
    led := TRUE;
  END_IF;
  IF atingiu AND led_estava_aceso THEN
    led := FALSE;
  END_IF;
  IF botao THEN
    led := TRUE;
  END_IF;
END_PROGRAM

CONFIGURATION Config0
  RESOURCE Res0 ON PLC
    TASK task0(INTERVAL := T#20ms, PRIORITY := 0);
    PROGRAM instance0 WITH task0 : prog0;
  END_RESOURCE
END_CONFIGURATION

(* ---- variante_j_pv12_pulso_antes_iniTRUE_realinhaFALSE.st ---- *)
(* Variante J (orquestrador, 2026-09-16): PV=12, pulso realinhado ao atingir o
   limite; ordem=pulso_antes, pulso inicial=TRUE, valor de realinhamento=FALSE. *)
PROGRAM prog0
  VAR
    botao AT %IX0.0 : BOOL;
    led   AT %QX0.0 : BOOL;
  END_VAR
  VAR
    pulso            : BOOL := TRUE;
    reset_ctu        : BOOL;
    atingiu          : BOOL;
    led_estava_aceso : BOOL;
    ctu0             : CTU;
  END_VAR

  pulso := NOT pulso;
  ctu0(CU := pulso, R := reset_ctu, PV := 12);
  atingiu := ctu0.Q;
  IF atingiu THEN
    pulso := FALSE;
  END_IF;
  reset_ctu := atingiu;
  led_estava_aceso := led;
  IF atingiu AND NOT led_estava_aceso THEN
    led := TRUE;
  END_IF;
  IF atingiu AND led_estava_aceso THEN
    led := FALSE;
  END_IF;
  IF botao THEN
    led := TRUE;
  END_IF;
END_PROGRAM

CONFIGURATION Config0
  RESOURCE Res0 ON PLC
    TASK task0(INTERVAL := T#20ms, PRIORITY := 0);
    PROGRAM instance0 WITH task0 : prog0;
  END_RESOURCE
END_CONFIGURATION

(* ---- variante_j_pv12_pulso_antes_iniTRUE_realinhaTRUE.st ---- *)
(* Variante J (orquestrador, 2026-09-16): PV=12, pulso realinhado ao atingir o
   limite; ordem=pulso_antes, pulso inicial=TRUE, valor de realinhamento=TRUE. *)
PROGRAM prog0
  VAR
    botao AT %IX0.0 : BOOL;
    led   AT %QX0.0 : BOOL;
  END_VAR
  VAR
    pulso            : BOOL := TRUE;
    reset_ctu        : BOOL;
    atingiu          : BOOL;
    led_estava_aceso : BOOL;
    ctu0             : CTU;
  END_VAR

  pulso := NOT pulso;
  ctu0(CU := pulso, R := reset_ctu, PV := 12);
  atingiu := ctu0.Q;
  IF atingiu THEN
    pulso := TRUE;
  END_IF;
  reset_ctu := atingiu;
  led_estava_aceso := led;
  IF atingiu AND NOT led_estava_aceso THEN
    led := TRUE;
  END_IF;
  IF atingiu AND led_estava_aceso THEN
    led := FALSE;
  END_IF;
  IF botao THEN
    led := TRUE;
  END_IF;
END_PROGRAM

CONFIGURATION Config0
  RESOURCE Res0 ON PLC
    TASK task0(INTERVAL := T#20ms, PRIORITY := 0);
    PROGRAM instance0 WITH task0 : prog0;
  END_RESOURCE
END_CONFIGURATION

(* ---- variante_k_pv12_ctu_antes_iniFALSE_led_atrasado.st ---- *)
(* Variante K (orquestrador, 2026-09-16): PV=12, pulso realinhado ao atingir o
   limite; ordem=ctu_antes, pulso inicial=FALSE, realinhamento=FALSE; LED alterna com o limite atrasado 1 ciclo (reset_ctu). *)
PROGRAM prog0
  VAR
    botao AT %IX0.0 : BOOL;
    led   AT %QX0.0 : BOOL;
  END_VAR
  VAR
    pulso            : BOOL := FALSE;
    reset_ctu        : BOOL;
    atingiu          : BOOL;
    led_estava_aceso : BOOL;
    ctu0             : CTU;
  END_VAR

  ctu0(CU := pulso, R := reset_ctu, PV := 12);
  atingiu := ctu0.Q;
  IF atingiu THEN
    pulso := FALSE;
  END_IF;
  pulso := NOT pulso;
  led_estava_aceso := led;
  IF reset_ctu AND NOT led_estava_aceso THEN
    led := TRUE;
  END_IF;
  IF reset_ctu AND led_estava_aceso THEN
    led := FALSE;
  END_IF;
  reset_ctu := atingiu;
  IF botao THEN
    led := TRUE;
  END_IF;
END_PROGRAM

CONFIGURATION Config0
  RESOURCE Res0 ON PLC
    TASK task0(INTERVAL := T#20ms, PRIORITY := 0);
    PROGRAM instance0 WITH task0 : prog0;
  END_RESOURCE
END_CONFIGURATION

(* ---- variante_k_pv12_pulso_antes_iniTRUE_led_atrasado.st ---- *)
(* Variante K (orquestrador, 2026-09-16): PV=12, pulso realinhado ao atingir o
   limite; ordem=pulso_antes, pulso inicial=TRUE, realinhamento=FALSE; LED alterna com o limite atrasado 1 ciclo (reset_ctu). *)
PROGRAM prog0
  VAR
    botao AT %IX0.0 : BOOL;
    led   AT %QX0.0 : BOOL;
  END_VAR
  VAR
    pulso            : BOOL := TRUE;
    reset_ctu        : BOOL;
    atingiu          : BOOL;
    led_estava_aceso : BOOL;
    ctu0             : CTU;
  END_VAR

  pulso := NOT pulso;
  ctu0(CU := pulso, R := reset_ctu, PV := 12);
  atingiu := ctu0.Q;
  IF atingiu THEN
    pulso := FALSE;
  END_IF;
  led_estava_aceso := led;
  IF reset_ctu AND NOT led_estava_aceso THEN
    led := TRUE;
  END_IF;
  IF reset_ctu AND led_estava_aceso THEN
    led := FALSE;
  END_IF;
  reset_ctu := atingiu;
  IF botao THEN
    led := TRUE;
  END_IF;
END_PROGRAM

CONFIGURATION Config0
  RESOURCE Res0 ON PLC
    TASK task0(INTERVAL := T#20ms, PRIORITY := 0);
    PROGRAM instance0 WITH task0 : prog0;
  END_RESOURCE
END_CONFIGURATION
